FUNCTION_BLOCK FB_Math
VAR
	calls : INT;
END_VAR

{attribute 'TcRpcEnable'}
METHOD Addition
VAR_INPUT
	a: DINT;
	b: DINT;
END_VAR
VAR_OUTPUT
	sum: DINT;
END_VAR
sum := a + b;
calls := calls + 1;
END_METHOD

END_FUNCTION_BLOCK

(* stored: Version 1.1.0.1, ProductVersion 3.1.0.26
   POU FB_Math: Id {08e5cb93-d3b0-4799-8ac9-227213fd8810}
   Method Addition: Id {e1bdf1e4-5f4f-4c5b-9be7-6c14ec4d4362} *)
